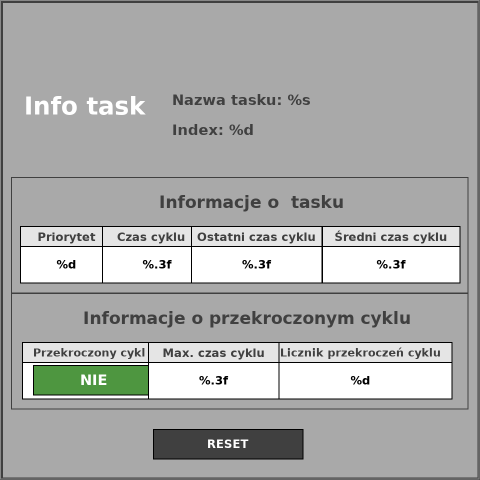
VISUALIZATION PH_TaskInfo  // 480x480
VAR_IN_OUT
	fbTaskInfo								: FB_TaskInfo;
	bReset									: BOOL;
END_VAR
VAR

END_VAR
    Rectangle (0,0 480x480)
    Label (21,91 150x30), "Info task"
    RoundedRectangle (11,177 457x116)
    Label (156,187 185x30), "Informacje o tasku"
    Rectangle (169,85 307x30), "Nazwa tasku: %s", text variable: fbTaskInfo.sTaskName
    Rectangle (169,115 150x30), "Index: %d", text variable: fbTaskInfo.byIndex
    RoundedRectangle (11,293 457x116)
    Label (80,303 320x30), "Informacje o przekroczonym cyklu"
    Group (20,226 82x57)
        RoundedRectangle (0,0 93x22), "Priorytet"
        Rectangle (0,20 93x37), "%d", text variable: fbTaskInfo.uiPriority
    RoundedRectangle (20,226 93x22), "Priorytet"
    Rectangle (20,246 93x37), "%d", text variable: fbTaskInfo.uiPriority
    Group (269,342 183x57)
        RoundedRectangle (0,0 183x22), "Licznik przekroczeń cyklu"
        Rectangle (0,20 183x37), "%d", text variable: fbTaskInfo.udiCountExceedCycle
    RoundedRectangle (269,342 183x22), "Licznik przekroczeń cyklu"
    Rectangle (269,362 183x37), "%d", text variable: fbTaskInfo.udiCountExceedCycle
    Group (22,342 126x57)
        RoundedRectangle (0,0 144x22), "Przekroczony cykl"
        Rectangle (0,20 144x37)
        RoundedRectangle (11,23 122x30), "TAK"
        RoundedRectangle (11,23 122x30), "NIE", invisible if: fbTaskInfo.bCycleTimeExceeded
    RoundedRectangle (22,342 144x22), "Przekroczony cykl"
    Rectangle (22,362 144x37)
    RoundedRectangle (33,365 122x30), "TAK"
    RoundedRectangle (33,365 122x30), "NIE", invisible if: fbTaskInfo.bCycleTimeExceeded
    Group (102,226 89x57)
        RoundedRectangle (0,0 110x22), "Czas cyklu"
        Rectangle (0,20 110x37), "%.3f", text variable: fbTaskInfo.rCycleTime
    RoundedRectangle (102,226 110x22), "Czas cyklu"
    Rectangle (102,246 110x37), "%.3f", text variable: fbTaskInfo.rCycleTime
    Group (191,226 131x57)
        RoundedRectangle (0,0 131x22), "Ostatni czas cyklu"
        Rectangle (0,20 131x37), "%.3f", text variable: fbTaskInfo.rLastExecTime
    RoundedRectangle (191,226 131x22), "Ostatni czas cyklu"
    Rectangle (191,246 131x37), "%.3f", text variable: fbTaskInfo.rLastExecTime
    Group (322,226 128x57)
        RoundedRectangle (0,0 138x22), "Średni czas cyklu"
        Rectangle (0,20 138x37), "%.3f", text variable: fbTaskInfo.rAverageCycleTime
    RoundedRectangle (322,226 138x22), "Średni czas cyklu"
    Rectangle (322,246 138x37), "%.3f", text variable: fbTaskInfo.rAverageCycleTime
    Group (148,342 121x57)
        RoundedRectangle (0,0 131x22), "Max. czas cyklu"
        Rectangle (0,20 131x37), "%.3f", text variable: fbTaskInfo.rMaxExecTime
    RoundedRectangle (148,342 131x22), "Max. czas cyklu"
    Rectangle (148,362 131x37), "%.3f", text variable: fbTaskInfo.rMaxExecTime
    RoundedRectangle (153,429 150x30), "RESET", colour toggle: bReset
        tap bReset
END_VISUALIZATION

(* stored: Version 1.1.0.1, ProductVersion 3.1.4024.3
   Visu PH_TaskInfo: Id {b427f2cf-ee45-4b1a-8ab0-9133e5bc0b51} *)
